// TIA Portal V18 export
DATA_BLOCK "ServoV90_A1"   // DB2501
{ S7_Optimized_Access := 'FALSE' }
VERSION : 0.1
// stored: AutoNumber false, DBAccessibleFromOPCUA true, DBAccessibleFromWebserver true, IsOnlyStoredInLoadMemory false, IsWriteProtectedInAS false
   VAR RETAIN
      In : Struct
         iInterlock : Bool := TRUE;   // interlock
         "iManJog+" : Bool := FALSE;   // positive motion/action/...manually
         "iManJog-" : Bool := FALSE;   // negtive motion/action/...manually
         iAutoStart : Bool := FALSE;   // negtive motion/action/...automaticly
         iHome : Bool := FALSE;   // Homing
         iCancelTask : Bool := FALSE;   // Cancel task
         iPauseTask : Bool := FALSE;   // Pause task
         iManStart : Bool := FALSE;   // positive motion/action/...automaticly
         iManListStart : Bool := FALSE;
         iLimitSwitchActive : Bool := TRUE;
         iLimitSoftActive : Bool := TRUE;
         iRunningTimeout : Time := T#0MS;
         iHomingTimeout : Time := T#0MS;
         iAutoPosition : DInt := 0;
         iAutoVelocity : Int := 0;
         iManListPosition : DInt := 0;
         iManListVelocity : Int := 10000;
         iManListNumber : Int := 0;   // position list number
         iManPosition : DInt := 318250;
         iManVelocity : Int := 10000;
         iMode : Int := 0;   // 1-相对;2-绝对
      END_STRUCT;
      Out : Struct
         oReady : Bool := FALSE;
         oWarning : Bool := FALSE;   // warning
         oError : Bool := TRUE;   // error
         oInterlock : Bool := TRUE;
         oServoEnable : Bool := FALSE;
         oRunning : Bool := FALSE;
         oHoming : Bool := FALSE;
         oHomeRef : Bool := TRUE;
         oServoPosOK : Bool := FALSE;
         oErrorCode : Int := -244;
         oStatus : Int := 0;
         oActPosition : DInt := 93294;
         oManualListPos : DInt := 3419;
      END_STRUCT;
      IO : Struct
         ioManEnale : Bool := FALSE;
         ioAutoEnale : Bool := FALSE;
      END_STRUCT;
      Spare : Struct
         S : Array[0..100] of Byte;
      END_STRUCT;
      Manual : Struct
         Index : Int := 1;
         Pos : Array[1..20] of Struct
            Pos : DInt;
            Vel : Int;
         END_STRUCT;
      END_STRUCT;
      Auto : Struct
         Index : Int := 6;
         Pos : Array[1..20] of Struct
            Pos : DInt;
            Vel : Int;
         END_STRUCT;
      END_STRUCT;
      Interlock : Struct
         Active : Bool := FALSE;
         Case1 : Bool := TRUE;
         Case2 : Bool := TRUE;
         Case3 : Bool := FALSE;
         Case4 : Bool := FALSE;
         Case5 : Bool := FALSE;
         Case6 : Bool := FALSE;
         Case7 : Bool := FALSE;
         Case8 : Bool := FALSE;
         Case9 : Bool := FALSE;
         Case10 : Bool := FALSE;
      END_STRUCT;
      PositionOk : Array[1..20] of Bool;
      Home_Pos : Struct
         "Home Pos Pls" : Bool := FALSE;
         "Arrow indication" : Int := 0;
         "Process prompt" : Int := 0;
         "Button prompt" : Int := 0;
      END_STRUCT;
   END_VAR
BEGIN
   Spare.S[0..100] := 16#00;
   Manual.Pos[1].Pos := 3419;
   Manual.Pos[2].Pos := 48386;
   Manual.Pos[3].Pos := 93294;
   Manual.Pos[4].Pos := 138335;
   Manual.Pos[5].Pos := 183464;
   Manual.Pos[6].Pos := 228443;
   Manual.Pos[7].Pos := 273535;
   Manual.Pos[8].Pos := 318250;
   Manual.Pos[9..20].Pos := 0;
   Manual.Pos[1..8].Vel := 10000;
   Manual.Pos[9..20].Vel := 0;
   Auto.Pos[1].Pos := 3419;
   Auto.Pos[2].Pos := 48386;
   Auto.Pos[3].Pos := 93294;
   Auto.Pos[4].Pos := 138335;
   Auto.Pos[5].Pos := 183464;
   Auto.Pos[6].Pos := 228443;
   Auto.Pos[7].Pos := 273535;
   Auto.Pos[8].Pos := 318250;
   Auto.Pos[9..20].Pos := 0;
   Auto.Pos[1..8].Vel := 10000;
   Auto.Pos[9..20].Vel := 0;
   // Auto.Pos[1] : 1.取料位置
   // Auto.Pos[2] : 2.放料位置
   // Auto.Pos[3] : 3.
   // Auto.Pos[4] : 4.
   // Auto.Pos[5] : 5.
   // Auto.Pos[6] : 6.
   // Auto.Pos[7] : 7.
   // Auto.Pos[8] : 8.
   // Auto.Pos[9] : 9.
   PositionOk[1] := FALSE;   // [1]
   PositionOk[2] := FALSE;   // [2]
   PositionOk[3] := FALSE;   // [3]
   PositionOk[4] := FALSE;   // [4]
   PositionOk[5] := FALSE;   // [5]
   PositionOk[6] := FALSE;   // [6]
   PositionOk[7] := FALSE;   // [7]
   PositionOk[8] := FALSE;   // [8]
   PositionOk[9] := FALSE;   // [9]
   PositionOk[10..20] := FALSE;
END_DATA_BLOCK
